(* PLC project Appliances, Actility iec61131 1.0.28, author Laurent Nicq *)
(* stored: creationDateTime 2013-06-10T10:05:45, version 1.1.2, modificationDateTime 2013-08-02T14:18:21 *)

FUNCTION_BLOCK Auto_OFF_Common
  VAR_INPUT
    AutoOFF_Input : BOOL;
    AutoOFF_Time : TIME;
  END_VAR
  VAR_OUTPUT
    AutoOFF_Out : BOOL;
  END_VAR
  VAR
    AutoOFF_Enable : BOOL := TRUE;
    AutoOFF_Elapsed : TIME;
    AutoOff_timer : TP;
  END_VAR

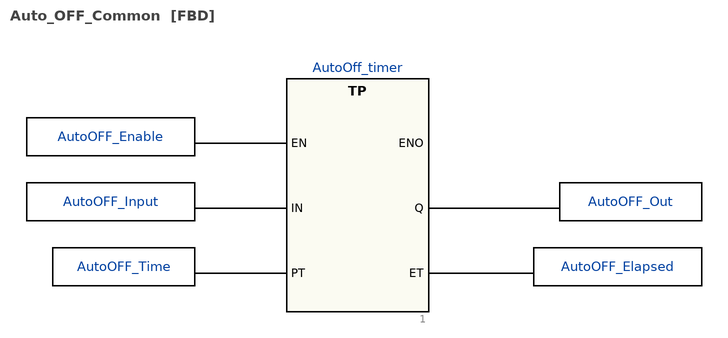
(* FBD diagram, written out as Structured Text *)
AutoOff_timer(EN := AutoOFF_Enable, IN := AutoOFF_Input, PT := AutoOFF_Time);
IF AutoOff_timer.ENO THEN AutoOFF_Out := AutoOff_timer.Q; END_IF;
IF AutoOff_timer.ENO THEN AutoOFF_Elapsed := AutoOff_timer.ET; END_IF;
END_FUNCTION_BLOCK

FUNCTION_BLOCK Auto_RESTART_Common
  VAR_INPUT
    AutoRESTART_Input : BOOL;
    AutoRESTART_Time : TIME;
  END_VAR
  VAR_OUTPUT
    AutoRESTART_Out : BOOL;
  END_VAR
  VAR
    AutoRESTART_Enable : BOOL := TRUE;
    AutoRESTART_Elapsed : TIME;
    AutoRestart_timer : TP;
  END_VAR
  VAR  (* added by the conversion: wires and edge detectors of the diagram *)
    _NOT12_OUT : BOOL;
    _NOT13_OUT : BOOL;
  END_VAR

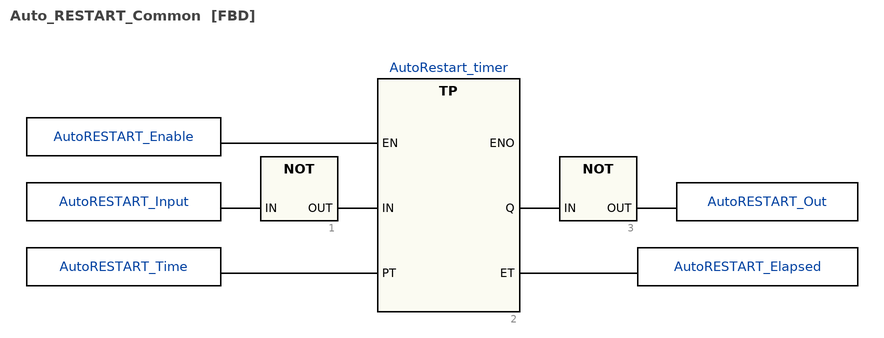
(* FBD diagram, written out as Structured Text *)
_NOT12_OUT := NOT AutoRESTART_Input;
AutoRestart_timer(EN := AutoRESTART_Enable, IN := _NOT12_OUT, PT := AutoRESTART_Time);
_NOT13_OUT := NOT AutoRestart_timer.Q;
AutoRESTART_Out := _NOT13_OUT;
IF AutoRestart_timer.ENO THEN AutoRESTART_Elapsed := AutoRestart_timer.ET; END_IF;
END_FUNCTION_BLOCK

PROGRAM Automatic_Appliance
  VAR_EXTERNAL
    Appliance1_State : BOOL;
    Appliance2_State : BOOL;
    Appliance1_Out : BOOL;
    Appliance2_Out : BOOL;
  END_VAR
  VAR
    Time_AutoOff : TIME := T#10s;
    Time_AutoRestart : TIME := T#20s;
    Auto_OFF_Test : Auto_OFF_Common;
    Auto_RESTART_Test : Auto_RESTART_Common;
  END_VAR

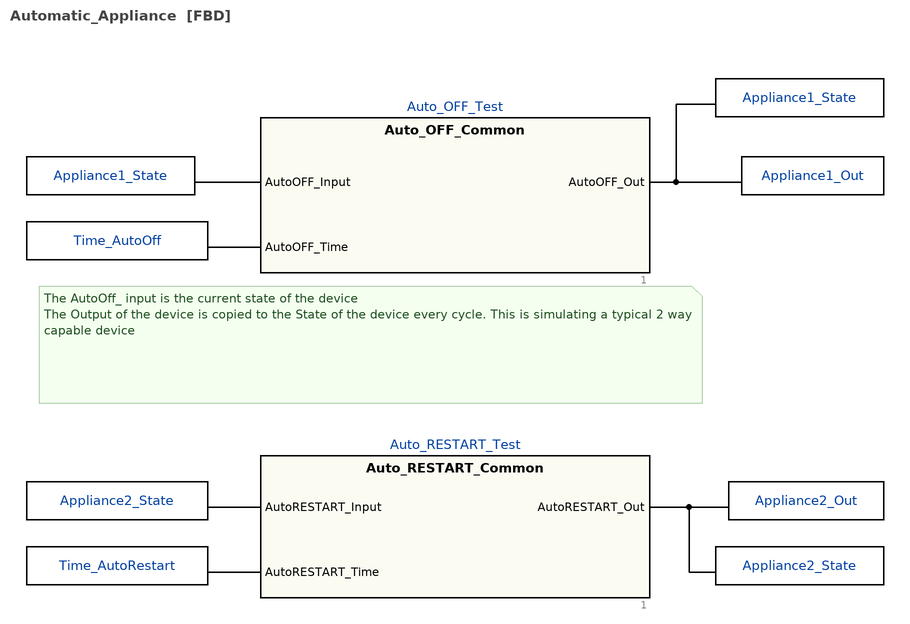
(* FBD diagram, written out as Structured Text *)
Auto_OFF_Test(AutoOFF_Input := Appliance1_State, AutoOFF_Time := Time_AutoOff);
(* The AutoOff_ input is the current state of the device
The Output of the device is copied to the State of the device every cycle. This is simulating a typical 2 way capable device *)
Auto_RESTART_Test(AutoRESTART_Input := Appliance2_State, AutoRESTART_Time := Time_AutoRestart);
Appliance1_State := Auto_OFF_Test.AutoOFF_Out;
Appliance1_Out := Auto_OFF_Test.AutoOFF_Out;
Appliance2_Out := Auto_RESTART_Test.AutoRESTART_Out;
Appliance2_State := Auto_RESTART_Test.AutoRESTART_Out;
END_PROGRAM

FUNCTION_BLOCK Auto_Light_Common
  VAR_INPUT
    Light_Motion_Detected : BOOL;
    Light_State : BOOL;
  END_VAR
  VAR_OUTPUT
    Light_Output : BOOL;
  END_VAR
  VAR
    Light_Auto_Enable : BOOL := TRUE;  (* Not used yet by IEC engine *)
    Light_ON_Elapsed : TIME;
  END_VAR
  VAR_INPUT
    Light_ON_Timer1 : TIME;
    Light_ON_Timer2 : TIME;
  END_VAR
  VAR
    Light_ON_Timer : TP;
  END_VAR
  VAR_INPUT
    Light_ON_Timer_Select : BOOL;  (* False: Short Time True: long Time *)
    Light_ON_Level : DINT := 50;  (* Detection Light level from 0% to 100% *)
    Current_Light_Level : DINT := 100;  (* Measured Light level from 0% to 100% *)
  END_VAR
  VAR
    Rising_Edge : R_TRIG;
  END_VAR
  VAR  (* added by the conversion: wires and edge detectors of the diagram *)
    _NOT23_OUT : BOOL;
    _LE20_OUT : BOOL;
    _AND15_OUT : BOOL;
    _SEL16_OUT : TIME;
  END_VAR

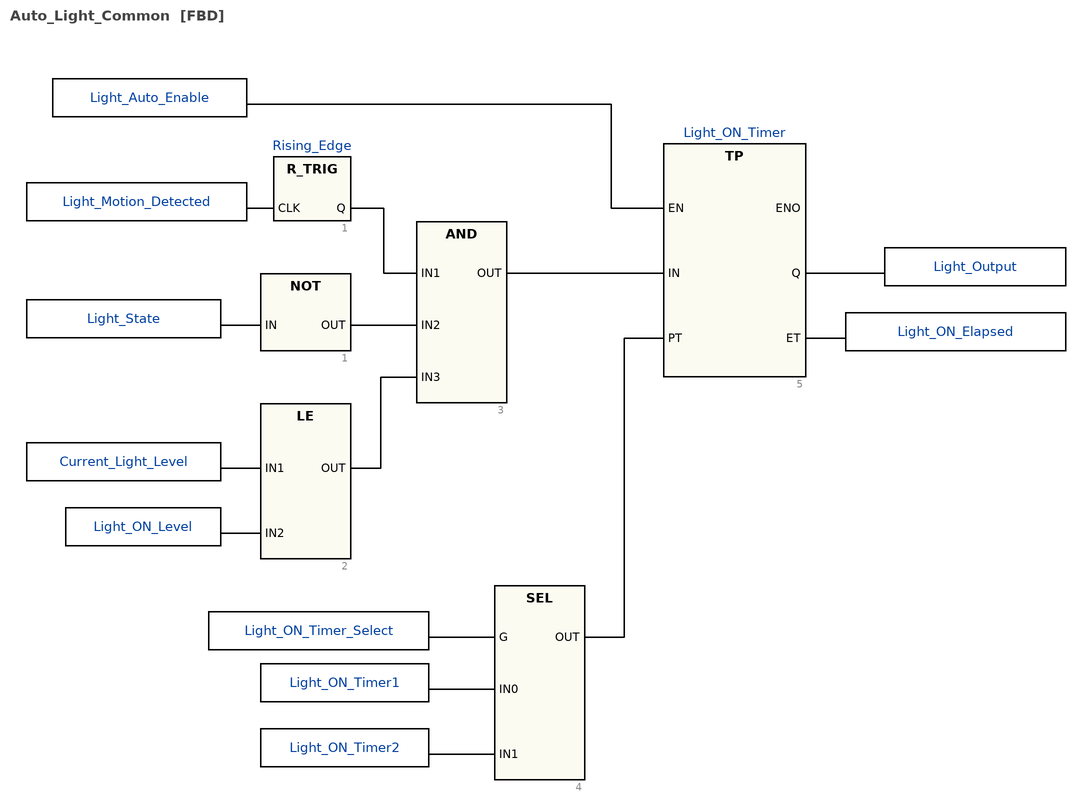
(* FBD diagram, written out as Structured Text *)
Rising_Edge(CLK := Light_Motion_Detected);
_NOT23_OUT := NOT Light_State;
_LE20_OUT := Current_Light_Level <= Light_ON_Level;
_AND15_OUT := Rising_Edge.Q AND _NOT23_OUT AND _LE20_OUT;
_SEL16_OUT := SEL(Light_ON_Timer_Select, Light_ON_Timer1, Light_ON_Timer2);
Light_ON_Timer(EN := Light_Auto_Enable, IN := _AND15_OUT, PT := _SEL16_OUT);
IF Light_ON_Timer.ENO THEN Light_Output := Light_ON_Timer.Q; END_IF;
IF Light_ON_Timer.ENO THEN Light_ON_Elapsed := Light_ON_Timer.ET; END_IF;
END_FUNCTION_BLOCK

PROGRAM Automatic_Light
  VAR
    Auto_Light_Test : Auto_Light_Common;
    Motion_Simul : BOOL;
    Light_State1 : BOOL;
    Light_Out1 : BOOL;
    Light_Timer_Select : BOOL := FALSE;
    Light_Timer1 : TIME := t#10s;
    Light_Timer2 : TIME := t#20s;
    Light_Level_Threshold : DINT := 50;
    Light_Level_Current : DINT := 49;
  END_VAR

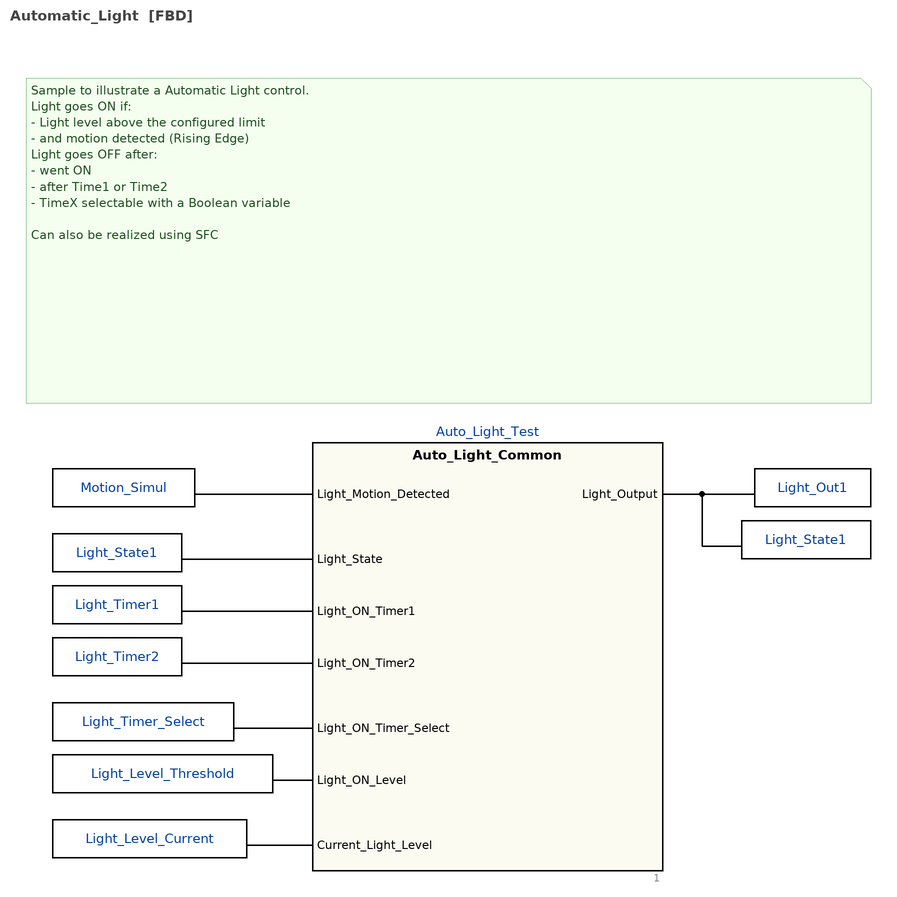
(* FBD diagram, written out as Structured Text *)
(* Sample to illustrate a Automatic Light control.
Light goes ON if:
 - Light level above the configured limit
 - and motion detected (Rising Edge)
Light goes OFF after:
 - went ON
 - after Time1 or Time2
 - TimeX selectable with a Boolean variable

Can also be realized using SFC *)
Auto_Light_Test(Light_Motion_Detected := Motion_Simul, Light_State := Light_State1, Light_ON_Timer1 := Light_Timer1, Light_ON_Timer2 := Light_Timer2, Light_ON_Timer_Select := Light_Timer_Select, Light_ON_Level := Light_Level_Threshold, Current_Light_Level := Light_Level_Current);
Light_Out1 := Auto_Light_Test.Light_Output;
Light_State1 := Auto_Light_Test.Light_Output;
END_PROGRAM

CONFIGURATION config
  RESOURCE resource_main ON PLC
    VAR_GLOBAL
      Appliance1_Out AT %QX1.0 : BOOL;
      Appliance1_State AT %IX1.0 : BOOL;
      Appliance2_Out AT %QX2.0 : BOOL;
      Appliance2_State AT %IX2.0 : BOOL;
    END_VAR
    TASK Sampling(INTERVAL := T#1s, PRIORITY := 0);
    PROGRAM Light WITH Sampling : Automatic_Light;
    PROGRAM Appliance WITH Sampling : Automatic_Appliance;
  END_RESOURCE
END_CONFIGURATION
